TYPE "HU_Tank_HMI"
VERSION : 0.1
// Block: HU_Tank_HMI
   STRUCT
      Alarm : Bool;
      RecirculationPump_Running : Bool;
      HeatExchangerFan_Running : Bool;
      HeatingUnit1_Running : Bool;
      HeatingUnit2_Running : Bool;
      EvChillerWater : Bool;
      OilTemperature : Real;
      WaterTemperature : Real;
      WeeklyClockEnabled : Real;
   END_STRUCT;

END_TYPE
